TYPE EtcSlaveBase_82538BE2 :
STRUCT
END_STRUCT
END_TYPE

(* stored: Version 1.2.0.0, ProductVersion 3.1.4024.9
   DUT EtcSlaveBase_82538BE2: Id {cd426701-a7ea-4c49-a007-c258741191ce} *)
